(* IEC 61131-3 sources: ArfBotOS/Codesys-4/ArfBotOS.fbsdev/Application.iecapp^/FUN/pause, 2 files *)

(* ---- F_BuildPauseCmd.fn.st ---- *)
FUNCTION F_BuildPauseCmd : STRING(GVL_App.COMMAND_LEN)
VAR_INPUT
	stCommand: ST_PauseCmd;
END_VAR
VAR
    _Command: STRING(GVL_App.COMMAND_LEN);
END_VAR
VAR CONSTANT
	_Delimiter: STRING:=' ';
END_VAR

// clear the command
_Command:='';

// build command
F_AddElement(_Command, _Delimiter, TIME_TO_STRING(stCommand.PauseTime));

// set function equal to command
F_BuildPauseCmd := _Command;
END_FUNCTION

(* ---- FB_ParsePauseCmd.fb.st ---- *)
FUNCTION_BLOCK FB_ParsePauseCmd
VAR_INPUT
	Command: STRING(GVL_App.COMMAND_LEN);
END_VAR
VAR_OUTPUT
	stCommand: ST_PauseCmd;
	Error: BOOL;
	ErrorDescription: STRING;
END_VAR
VAR
	_CmdParams: ARRAY [0..GVL_App.COMMAND_LEN] OF STRING;
END_VAR

// T#30s

Error:=FALSE;
ErrorDescription:='';

// split command string into commands
_CmdParams:=F_SplitCmd(Command:=Command);

stCommand.PauseTime := STRING_TO_TIME(_CmdParams[0]);
END_FUNCTION_BLOCK
